// TIA Portal V17 export
// export: Created 2024-01-30T08:49:14.3089565Z, ExportSetting WithDefaults, DisplayName Totally Integrated Automation Portal, DisplayVersion V17 Update 6, DisplayName TIA Portal Openness, DisplayVersion V17 Update 6, DisplayName TIA Portal Version Control Interface, DisplayVersion V17, DisplayName STEP 7 Professional, DisplayVersion V17 Update 6, DisplayName STEP 7 Safety, DisplayVersion V17 Update 6, DisplayName WinCC Advanced, DisplayVersion V17 Update 6
DATA_BLOCK "DB_CMMT_ST"   // DB13
{ S7_Optimized_Access := 'TRUE' }
VERSION : 0.1
// stored: AutoNumber true, DBAccessibleFromOPCUA true, DBAccessibleFromWebserver true, IsOnlyStoredInLoadMemory false, IsRetainMemResEnabled false, IsWriteProtectedInAS false, MemoryReserve 100
   VAR
      "PLC -> CMMT" : "UDT_FESTO_CMMT_IN";
      "CMMT -> PLC" { S7_SetPoint := 'True'} : "UDT_FESTO_CMMT_OUT";
      ActualPos_mm { S7_SetPoint := 'True'} : Real;
      AcutalVelocity_mm_s : Real;
      SetPosition_mm : Real;
      SetVelocity_mm_s : Real := 20.0;
      HMI : Struct
         Scaled_ActualPos : Real;
         Scaled_SetpointPosition : Real;
         Scaled_ActualVelocity : Real;
      END_STRUCT;
      CLAMPING_TORQUE : Struct
         Execute : Bool;
         LinearRotative : Bool;
         ClampingTorque : Real;
         PercentForce : Real;
      END_STRUCT;
      CMMT_ST_ErrorWarningMessage : String;
   END_VAR
BEGIN
   "PLC -> CMMT".CancelTraversing := TRUE;
   "PLC -> CMMT".IntermediateStop := TRUE;
   "PLC -> CMMT".OverV := 100;
   "PLC -> CMMT".BaseSpeedValue := 0.125;
END_DATA_BLOCK
